Staubli VAL3: onStart.pgx

public program onStart(string& x_sItem[] (dimensions=1))
  local string l_sType
  local num i
  local string l_sPath
begin
  // language
  call language2:getLanguage(l_sPath)
  if l_sPath!=language2:libPath()+"/"+saveData:language
    // set language
    call language2:setLanguage(language2:libPath()+"/"+saveData:language)
  endIf
end
